// TIA Portal V19 export
DATA_BLOCK "STRING"   // DB169
{ S7_Optimized_Access := 'FALSE' }
   VAR
      PRODUCT_NAME : String[50];
      BATCH_NO : String[50];
      EQUIPMENT_ID_NO : String[50];
      RECIPE_NO : String[50];
      OPERATOR_NAME : String[50];
      EMPLOYE_CODE : String[50];
   END_VAR
BEGIN
END_DATA_BLOCK
